FUNCTION_BLOCK FB_Dakraam
VAR_INPUT
END_VAR
VAR_OUTPUT
END_VAR
VAR
END_VAR

END_FUNCTION_BLOCK

(* stored: Version 1.1.0.1, ProductVersion 3.1.4024.12
   POU FB_Dakraam: Id {7824faf0-75c8-4105-b5d4-0ed7696b36b3}, SpecialFunc None *)
